FUNCTION_BLOCK FB_LoadCell
VAR_INPUT
END_VAR
VAR_OUTPUT
END_VAR
VAR
END_VAR

END_FUNCTION_BLOCK

(* stored: Version 1.1.0.1, ProductVersion 3.1.4024.10
   POU FB_LoadCell: Id {b088edfa-6b7c-432a-9854-207f4dd9976a}, SpecialFunc None *)
